(* CoDeSys 2.3.9.31 project: Block3.pro *)
(* Libraries: STANDARD.LIB 5.6.98 12:03:02 *)

(* Task configuration *)
TASK Standard (PRIORITY := 0, INTERVAL := T#5ms);
	MAIN
END_TASK

(* Global variable list: Global_Variables *)
VAR_GLOBAL
	btn_yellow AT %I* : BOOL;
	btn_blue AT %I* : BOOL;
	led_green AT %Q*: BOOL;
	led_red AT %Q*: BOOL;
END_VAR
VAR_GLOBAL CONSTANT
	CODESIZE : INT := 4;
END_VAR

(* Global variable list: TwinCAT_Configuration *)
(* Generated automatically by TwinCAT - (read only) *)
VAR_CONFIG
	.btn_yellow AT %IX4.0 : BOOL;	(*  ~ {LinkedWith:TIID^Device 1 (EtherCAT)^Term 1 (EK1200)^Term 2 (EL1004)^Channel 1^Input} *)
	.btn_blue AT %IX0.1 : BOOL;	(*  ~ {LinkedWith:TIID^Device 1 (EtherCAT)^Term 1 (EK1200)^Term 2 (EL1004)^Channel 2^Input} *)
	.led_green AT %QX0.0 : BOOL;	(*  ~ {LinkedWith:TIID^Device 1 (EtherCAT)^Term 1 (EK1200)^Term 3 (EL2004)^Channel 2^Output} *)
	.led_red AT %QX0.1 : BOOL;	(*  ~ {LinkedWith:TIID^Device 1 (EtherCAT)^Term 1 (EK1200)^Term 3 (EL2004)^Channel 1^Output} *)
END_VAR

(* Data type *)
TYPE ST_Tresor :
	(
		ST_init,
		ST_close,
		ST_wrong,
		ST_check,
		ST_open,
		ST_progInit,
		ST_prog,
		ST_progExit
);
END_TYPE

(* POU MAIN, ST *)
PROGRAM MAIN
VAR
	state : ST_Tresor;
	b_y : EdgeDetectorDouble;
	b_b : EdgeDetectorDouble;
	code : ARRAY[1..CODESIZE] OF BOOL;
	index : INT := 1;
	t_delay : INT := duration;
	flag_wrong : BOOL := FALSE;
END_VAR
VAR CONSTANT
	duration : INT := 1000;
END_VAR
b_y(inputValue := btn_yellow, threshold  := 30);
b_b(inputValue := btn_blue, threshold  := 30);
CASE state OF
	ST_init:
		state := ST_close;
		code[1] := TRUE;
		code[2] := TRUE;
		code[3] := FALSE;
		code[4] := TRUE;
	ST_close:
		led_green := FALSE;
		led_red := FALSE;
		index := 1;
		state := ST_check;
		flag_wrong := FALSE;
	ST_wrong:
		IF t_delay > 0THEN
			T_delay := T_delay - 1;
			led_red := TRUE;
		ELSE
			T_delay := duration;
			led_red := FALSE;
			state := ST_close;
		END_IF
	ST_check:
		IF b_b.risingEdge THEN
			IF code[index] = FALSE THEN
				flag_wrong := TRUE;
			END_IF
			index := index +1;
		ELSIF b_y.risingEdge THEN
			IF code[index] = TRUE THEN
				flag_wrong := TRUE;
			END_IF
			index := index +1;
		END_IF
		IF index > CODESIZE THEN
			IF flag_wrong = TRUE THEN
				state := ST_wrong;
				t_delay := duration;
			ELSE
				state := ST_open;
				t_delay := duration;
			END_IF
		END_IF
		IF b_b.double OR b_y.double THEN
			state := ST_close;
		END_IF
	ST_open:
		IF t_delay > 0THEN
			T_delay := T_delay - 1;
			led_green := TRUE;
		ELSE
			T_delay := duration;
			led_green := FALSE;
			state := ST_close;
		END_IF
		IF btn_yellow AND btn_blue THEN
			state := ST_progInit;
			t_delay := duration / 5;
		END_IF
	ST_progInit:
		t_delay := t_delay -1;
		led_green := TRUE;
		led_red := TRUE;
		IF t_delay = 0 THEN
			state := ST_prog;
			led_green := FALSE;
			led_red := FALSE;
			index := 1;
		END_IF
	ST_prog:
		IF b_b.risingEdge THEN
			code[index] := TRUE;
			index := index + 1;
		ELSIF b_y.risingEdge THEN
			code[index] := FALSE;
			index := index + 1;
		END_IF
		IF index > CODESIZE THEN
			state := ST_progExit;
			t_delay := duration / 5;
		END_IF
	ST_progExit:
		t_delay := t_delay -1;
		led_green := TRUE;
		led_red := TRUE;
		IF t_delay = 0 THEN
			state := ST_close;
		END_IF
END_CASE
END_PROGRAM

(* POU EdgeDetectorDouble, ST *)
FUNCTION_BLOCK EdgeDetectorDouble
VAR_INPUT
	inputValue : BOOL;
	threshold : INT;
END_VAR
VAR_OUTPUT
	risingEdge : BOOL;
	fallingEdge : BOOL;
	double : BOOL;
END_VAR
VAR
	prev : BOOL := FALSE;
	timer : INT := 0;
END_VAR
IF inputValue > prev THEN
	risingEdge := TRUE;
	fallingEdge := FALSE;
	IF timer < threshold THEN
		double := TRUE;
	ELSE
		double := FALSE;
	END_IF
	timer := 0;
ELSIF inputValue < prev THEN
	risingEdge := FALSE;
	fallingEdge := TRUE;
	IF timer < 32767 THEN
		timer := timer + 1;
	END_IF
	double := FALSE;
ELSE
	risingEdge := FALSE;
	fallingEdge := FALSE;
	IF timer < 32767 THEN
		timer := timer + 1;
	END_IF
	double := FALSE;
END_IF
prev := inputValue;
END_FUNCTION_BLOCK

(* POU EdgeDetector, ST *)
FUNCTION_BLOCK EdgeDetector
VAR_INPUT
	inputValue : BOOL;
END_VAR
VAR_OUTPUT
	risingEdge : BOOL;
	fallingEdge : BOOL;
END_VAR
VAR
	prev : BOOL := FALSE;
END_VAR
IF inputValue > prev THEN
	risingEdge := TRUE;
	fallingEdge := FALSE;
ELSIF inputValue < prev THEN
	risingEdge := FALSE;
	fallingEdge := TRUE;
ELSE
	risingEdge := FALSE;
	fallingEdge := FALSE;
END_IF
prev := inputValue;
END_FUNCTION_BLOCK
